// TIA Portal V19 export
VAR_GLOBAL   // PLC tag table "LB321"
   LB321_RullieraDopoTaglio_Pb_Aux2 AT %Q251.4 : Bool;   // 354SH2
   LB321_RullieraDopoTaglio_Pb_Aux1 AT %Q251.3 : Bool;   // 354SH1
   LB321_RullieraDopoTaglio_Lp_Aux2 AT %I252.0 : Bool;   // 354SH2
   LB321_RullieraDopoTaglio_Lp_Aux1 AT %I251.7 : Bool;   // 354SH1
END_VAR
